Staubli VAL3: reset.pgx

public program reset()
  local num l_nSize
  local num i
  local num l_nResult
  local string l_sKey
begin
  // reset it
  l_sKey="init"
  call onStart(l_sKey)
  // save it
  call save(l_nResult)
end
